// Block: PPrgArchive3

DATA_BLOCK PPrgArchive3
VERSION : 0.1
   NON_RETAIN
   VAR
      PRG : Array[201..300] of PPrg_Data;
   END_VAR

BEGIN
   // No initialization required
END_DATA_BLOCK
